# EPICS autosave request: iocBoot/iocsnd/auto_settings.req
file snd.req BL=$(BL),DEV=$(DEV),GROUP=G1
file snd.req BL=$(BL),DEV=$(DEV),GROUP=G2
